// TIA Portal V19 export
FUNCTION "FC_Modbus_ArduinoComms" : Void   // FC1, LAD
{ S7_Optimized_Access := 'TRUE' }
// stored: SetENOAutomatically false
BEGIN

REGION Network 1
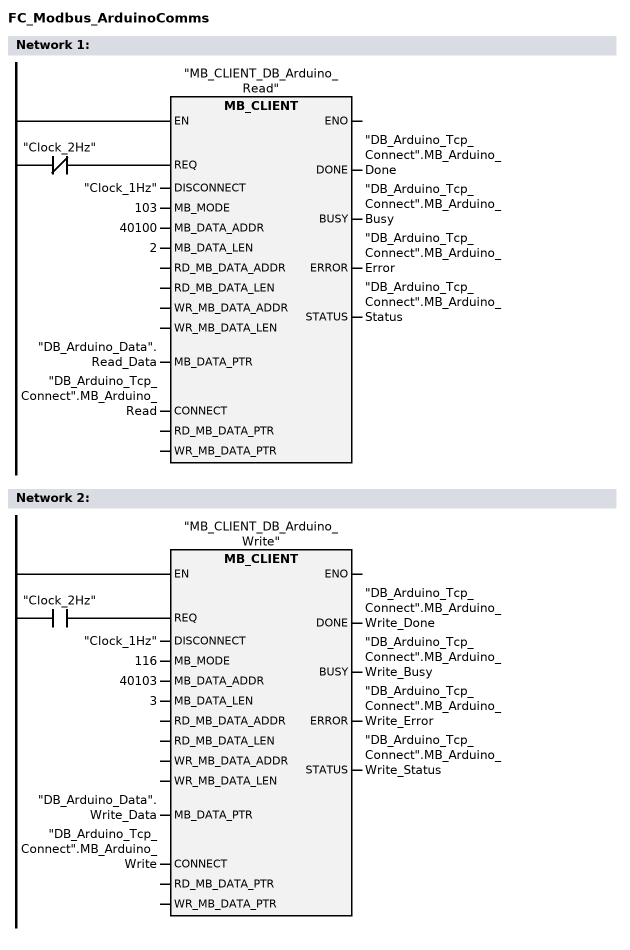
   RUNG wire#powerrail
      "MB_CLIENT_DB_Arduino_Read".MB_CLIENT(REQ := wire#w1, DISCONNECT := "Clock_1Hz", MB_MODE := 103, MB_DATA_ADDR := 40100, MB_DATA_LEN := 2, RD_MB_DATA_ADDR :=, RD_MB_DATA_LEN :=, WR_MB_DATA_ADDR :=, WR_MB_DATA_LEN :=, MB_DATA_PTR := "DB_Arduino_Data".Read_Data, CONNECT := "DB_Arduino_Tcp_Connect".MB_Arduino_Read, RD_MB_DATA_PTR :=, WR_MB_DATA_PTR :=, DONE => "DB_Arduino_Tcp_Connect".MB_Arduino_Done, BUSY => "DB_Arduino_Tcp_Connect".MB_Arduino_Busy, ERROR => "DB_Arduino_Tcp_Connect".MB_Arduino_Error, STATUS => "DB_Arduino_Tcp_Connect".MB_Arduino_Status)
   END_RUNG
   RUNG wire#powerrail
      I_Contact( "Clock_2Hz" )
   END_RUNG wire#w1
   // the same network as SCL:
   "MB_CLIENT_DB_Arduino_Read"(REQ := NOT "Clock_2Hz",   // MB_CLIENT
                           DISCONNECT := "Clock_1Hz",
                           MB_MODE := 103,
                           MB_DATA_ADDR := 40100,
                           MB_DATA_LEN := 2,
                           MB_DATA_PTR := "DB_Arduino_Data".Read_Data,
                           CONNECT := "DB_Arduino_Tcp_Connect".MB_Arduino_Read,
                           DONE => "DB_Arduino_Tcp_Connect".MB_Arduino_Done,
                           BUSY => "DB_Arduino_Tcp_Connect".MB_Arduino_Busy,
                           ERROR => "DB_Arduino_Tcp_Connect".MB_Arduino_Error,
                           STATUS => "DB_Arduino_Tcp_Connect".MB_Arduino_Status);
END_REGION

REGION Network 2
   RUNG wire#powerrail
      "MB_CLIENT_DB_Arduino_Write".MB_CLIENT(REQ := wire#w1, DISCONNECT := "Clock_1Hz", MB_MODE := 116, MB_DATA_ADDR := 40103, MB_DATA_LEN := 3, RD_MB_DATA_ADDR :=, RD_MB_DATA_LEN :=, WR_MB_DATA_ADDR :=, WR_MB_DATA_LEN :=, MB_DATA_PTR := "DB_Arduino_Data".Write_Data, CONNECT := "DB_Arduino_Tcp_Connect".MB_Arduino_Write, RD_MB_DATA_PTR :=, WR_MB_DATA_PTR :=, DONE => "DB_Arduino_Tcp_Connect".MB_Arduino_Write_Done, BUSY => "DB_Arduino_Tcp_Connect".MB_Arduino_Write_Busy, ERROR => "DB_Arduino_Tcp_Connect".MB_Arduino_Write_Error, STATUS => "DB_Arduino_Tcp_Connect".MB_Arduino_Write_Status)
   END_RUNG
   RUNG wire#powerrail
      Contact( "Clock_2Hz" )
   END_RUNG wire#w1
   // the same network as SCL:
   "MB_CLIENT_DB_Arduino_Write"(REQ := "Clock_2Hz",   // MB_CLIENT
                           DISCONNECT := "Clock_1Hz",
                           MB_MODE := 116,
                           MB_DATA_ADDR := 40103,
                           MB_DATA_LEN := 3,
                           MB_DATA_PTR := "DB_Arduino_Data".Write_Data,
                           CONNECT := "DB_Arduino_Tcp_Connect".MB_Arduino_Write,
                           DONE => "DB_Arduino_Tcp_Connect".MB_Arduino_Write_Done,
                           BUSY => "DB_Arduino_Tcp_Connect".MB_Arduino_Write_Busy,
                           ERROR => "DB_Arduino_Tcp_Connect".MB_Arduino_Write_Error,
                           STATUS => "DB_Arduino_Tcp_Connect".MB_Arduino_Write_Status);
END_REGION
END_FUNCTION
